FUNCTION_BLOCK Insertion //2d insertion that combines a slider (alignment) and screw (push)
VAR_INPUT
	enable : BOOL;
END_VAR
VAR_INPUT //interface references to existing drives
	slider : I_EncodedDrive;
	screw : I_ContinuousDrive;
END_VAR
VAR_OUTPUT
	contact AT %I* : BOOL;
	softContact : BOOL; //temporary
	
	busy : BOOL;
	error : BOOL;
	home : BOOL;
	
	homeSet : BOOL;
	
	sliderPos : LREAL;
END_VAR
(*
this FB encapsulates 2 drives into a generic insertion machine
the implementation of both drives should be called externally
an Insertion instance should be called in the scope it is declared in
*)

softContact := slider.contact AND screw.contact; //temporary

homeSet := slider.HomeSet AND screw.HomeSet;

busy := slider.Busy OR screw.Busy;
error := slider.Error OR screw.Error;
home := slider.AtHome AND screw.AtHome;

sliderPos := slider.CurrentPosition;

METHOD align : BOOL
VAR_INPUT
	targetPos : REAL;
END_VAR
slider.moveAbsolute(newTarget := targetPos);
END_METHOD

METHOD homingSequence : BOOL
VAR_INPUT
END_VAR
IF NOT slider.homeSet THEN
	slider.homingSequence();
END_IF

IF NOT screw.homeSet THEN
	screw.homingSequence();
END_IF

homingSequence := homeSet := slider.homeSet AND screw.homeSet;
END_METHOD

METHOD press : BOOL
VAR_INPUT
END_VAR
screw.moveContinuous(direction := MC_Negative_Direction);
END_METHOD

METHOD release : BOOL
VAR_INPUT
END_VAR
screw.moveContinuous(direction := MC_Positive_Direction);
END_METHOD

METHOD traverse : BOOL
VAR_INPUT
	direction : MC_Direction;
END_VAR
slider.moveContinuous(direction := MC_Negative_Direction);
END_METHOD

END_FUNCTION_BLOCK

(* stored: Version 1.1.0.1, ProductVersion 3.1.4024.11
   POU Insertion: Id {474cec8b-539b-4b97-8920-b045f392c812}, SpecialFunc None
   Method align: Id {150b5680-ccac-4b88-b9bd-ce3a432e6e4b}
   Method homingSequence: Id {1eff6ad7-4509-4cdc-81af-eef38809ec7f}
   Method press: Id {4b68a98e-5d52-4750-8c51-39e9aab9887f}
   Method release: Id {43664641-2403-4070-8d32-2915d9eeb09e}
   Method traverse: Id {2976ba6d-a5c4-4581-84e8-a5c41da415dd} *)
